SUBAPPLICATION Uebung_084 (* Beispiel für E_CYCLE *)
  (* Standard: 61499-2; Description: Copyright (c) 2023 Meisterschulen am Ostbahnhof This program and the accompanying materials are made available under the terms of the Eclipse Public License 2.0 which is available at https://www.eclipse.org/legal/epl-2.0/ SPDX-License-Identifier: EPL-2.0 *)
  (* Version 1.0, 2023-10-23, Franz Höpfinger, Meisterschulen am Ostbahnhof, initial API and implementation and/or initial documentation *)
  PACKAGE Uebungen;
  IMPORT logiBUS::io::DI::logiBUS_DI::Input_I1;
  IMPORT logiBUS::io::DI::logiBUS_DI::Input_I2;
  IMPORT logiBUS::io::DI::logiBUS_DI::Input_I3;
  IMPORT logiBUS::io::DI::logiBUS_DI_Events::BUTTON_SINGLE_CLICK;
  IMPORT logiBUS::io::DQ::logiBUS_DO::Output_Q1;
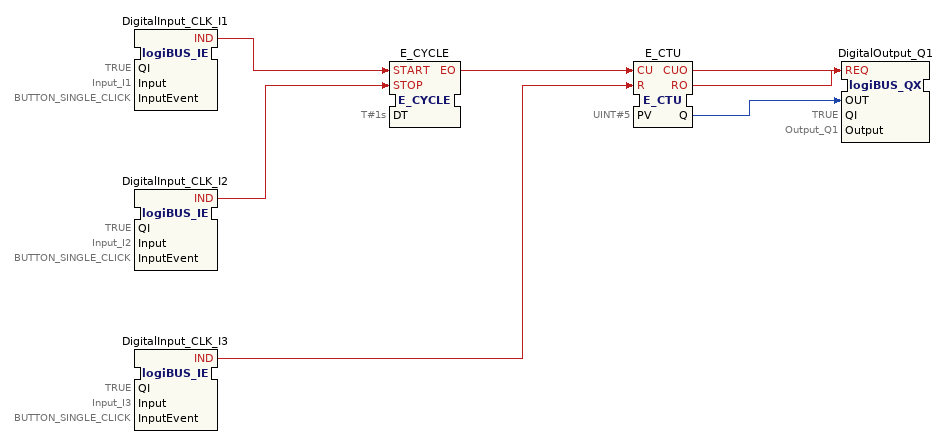
  FBS
    DigitalOutput_Q1 : logiBUS::io::DQ::logiBUS_QX(QI := TRUE, Output := Output_Q1);
    E_CTU : iec61499::events::E_CTU(PV := UINT#5);
    E_CYCLE : iec61499::events::E_CYCLE(DT := T#1s);
    DigitalInput_CLK_I2 : logiBUS::io::DI::logiBUS_IE(QI := TRUE, Input := Input_I2, InputEvent := BUTTON_SINGLE_CLICK);
    DigitalInput_CLK_I3 : logiBUS::io::DI::logiBUS_IE(QI := TRUE, Input := Input_I3, InputEvent := BUTTON_SINGLE_CLICK);
    DigitalInput_CLK_I1 : logiBUS::io::DI::logiBUS_IE(QI := TRUE, Input := Input_I1, InputEvent := BUTTON_SINGLE_CLICK);
  END_FBS
  EVENT_CONNECTIONS
    E_CTU.CUO TO DigitalOutput_Q1.REQ;
    E_CTU.RO TO DigitalOutput_Q1.REQ;
    E_CYCLE.EO TO E_CTU.CU;
    DigitalInput_CLK_I1.IND TO E_CYCLE.START;
    DigitalInput_CLK_I2.IND TO E_CYCLE.STOP;
    DigitalInput_CLK_I3.IND TO E_CTU.R;
  END_CONNECTIONS
  DATA_CONNECTIONS
    E_CTU.Q TO DigitalOutput_Q1.OUT;
  END_CONNECTIONS
END_SUBAPPLICATION
